{attribute 'qualified_only' := ''}
{attribute 'strict' := ''}
TYPE eFirmerVendorEvent1 :
(
	eNoInfo := 0,
	ePowerCurtailmentFromExternalCommand := 1,
	ePowerLimitationFromFrequencyWatt := 2,
	ePowerLimitationFromHighAverageGridVoltage := 3,
	ePowerLimitationFromAntiIslandingProtection := 4,
	ePowerLimitationFromGridCurrentRatingLimitation := 5,
	ePowerLimitationForHighTemperature := 6,
	ePowerLimitationForHighDCVoltage := 7,
	ePowerLimitationFromRampRateConnectionRamp := 9,
	ePowerLimitationFromMomentaryCessation := 10,
	ePowerLimitationFromRampRateNormalRampUp := 11,
	ePowerLimitationFromVoltWatt := 12,
	ePowerLimitationFromCapabilityRating := 13
);
END_TYPE

(* stored: Version 1.1.0.1, ProductVersion 3.1.4024.11
   DUT eFirmerVendorEvent1: Id {d63bd406-d577-4915-90bc-07cc2c4e13fa} *)
